// TwinCAT 3 PLC project TwinCat
// ProgramVersion: 3.1.4026.14
// libraries:
//   Tc2_Standard, * (Beckhoff Automation GmbH)
//   Tc2_System, * (Beckhoff Automation GmbH)
//   Tc3_Module, * (Beckhoff Automation GmbH)
// project tree:
//   DUTs/POUs/TEMPLATE ST FB%27s/ AdvancedFaultDetection.TcPOU (not stored), Auto_Manual_CycleControl.TcPOU (not stored), CYL.TcPOU (not stored), FB_analog.TcPOU (not stored), FB_Conveyor.TcPOU (not stored), FB_Fan.TcPOU (not stored), FB_FaultDetection.TcPOU (not stored), FB_FlowMeter.TcPOU (not stored), FB_IO_Card_ARRAY.TcPOU (not stored), FB_IO_CARD_BOOL.TcPOU (not stored), FB_LevelSensor.TcPOU (not stored), FB_Pump.TcPOU (not stored), FB_SensorHandler.TcPOU (not stored), FB_StackLight.TcPOU (not stored), FB_STATUS.TcPOU (not stored), FB_Tank.TcPOU (not stored), FB_Valve.TcPOU (not stored), FB_Valve_Proportional.TcPOU (not stored), FB_VFD_FWD_REV.TcPOU (not stored), Reject_Conveyor.TcPOU (not stored), SensorProcessing.TcPOU (not stored)
//   / PlcTask.TcTTO
//   POUs/ MAIN.TcPOU, POU.TcPOU
// real-time tasks:
//   TASK PlcTask: cycle T#10ms, priority 20, ADS port 350
//   TASK Job Task: cycle default, priority 32
//   TASK MC-Task (MET): cycle T#2ms, priority 3, ADS port 521
//   TASK MC-Task (MPT): cycle T#10ms, priority 8, ADS port 531

CONFIGURATION TwinCat
    RESOURCE PLC ON TwinCAT3
        TASK PlcTask(INTERVAL := T#10ms, PRIORITY := 20);
        PROGRAM MAIN WITH PlcTask : MAIN;
        PROGRAM POU WITH PlcTask : POU;
    END_RESOURCE
END_CONFIGURATION

// ---- POUs/MAIN.TcPOU
PROGRAM MAIN
VAR
  Main : BOOL;
  
END_VAR

END_PROGRAM

// ---- POUs/POU.TcPOU
PROGRAM POU
VAR
	Mode: BOOL;
	Fan_speed: REAL;
	STATUS: BOOL;
	Manual: BOOL;
	Fan_0: FB_Fan;
	SETPOINT: REAL := 15;
	CURRNET: REAL := 10;
	STARTMAN: BOOL;
	STOPMAN: BOOL;
	STARTAUTO: BOOL;
	STOPAUTO: BOOL;
	EMERGSTOP: BOOL;
	FAULT: BOOL;
	CYCLERUN: BOOL;
	FAULT_LOG: STRING;
	DELAY_TIMER: TON;
	START_DELAY: TON;
	EMERGSTOP_STATUS: BOOL;
	BUZZER: BOOL;
	MODESELECT: INT;
	STOPDELAY: TIME;
	STARTDELAY: TIME;
	FB_SensorHandler_0: FB_SensorHandler;
	SESNORSTATUS: BOOL;
	INPUT: BOOL;
	OUTPUT: BOOL;
	FAULTSTATUS: STRING(50);
END_VAR

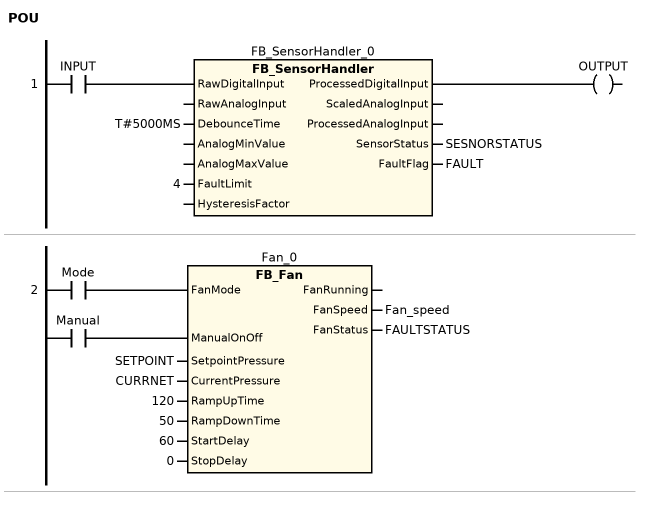
// NETWORK 1
FB_SensorHandler_0(
    RawDigitalInput := INPUT,
    DebounceTime := T#5000MS,
    FaultLimit := 4,
    SensorStatus => SESNORSTATUS,
    FaultFlag => FAULT); // FB_SensorHandler
OUTPUT := FB_SensorHandler_0.ProcessedDigitalInput;

// NETWORK 2
Fan_0(
    FanMode := Mode,
    ManualOnOff := Manual,
    SetpointPressure := SETPOINT,
    CurrentPressure := CURRNET,
    RampUpTime := 120,
    RampDownTime := 50,
    StartDelay := 60,
    StopDelay := 0,
    FanSpeed => Fan_speed,
    FanStatus => FAULTSTATUS); // FB_Fan

END_PROGRAM
